{attribute 'linkalways'} 
{attribute 'no_explicit_call' := 'This FB is a CLASS and must be accessed using methods or properties'}
{attribute 'enable_dynamic_creation'}
FUNCTION_BLOCK FINAL NE_DINT EXTENDS Node
VAR
	in1 : _DINT(0);
	in2 : _DINT(0);
	out : _BOOL(FALSE);
END_VAR

METHOD PUBLIC Clone : I_Node
VAR
	pNode : POINTER TO NE_DINT;
END_VAR
pNode := __NEW(NE_DINT);
Clone := pNode^;
END_METHOD

METHOD FB_init : BOOL
VAR_INPUT
	bInitRetains : BOOL; // if TRUE, the retain variables are initialized (warm start / cold start)
	bInCopyCode : BOOL;  // if TRUE, the instance afterwards gets moved into the copy code (online change)
END_VAR
AddInput('in1',THIS^.in1);
AddInput('in2',THIS^.in2);
AddOutput('out', THIS^.out);
END_METHOD

METHOD PROTECTED OnExecute
VAR
END_VAR
out.Value := in1.Value <> in2.Value;
END_METHOD

END_FUNCTION_BLOCK

(* stored: Version 1.1.0.1, ProductVersion 3.1.4024.15
   POU NE_DINT: Id {dc90bf6d-96e3-4071-902f-2370f234dd21}, SpecialFunc None
   Folder Constructor: Id {d7f0702d-e194-47fb-881f-41a2618626ac}
   Method Clone: Id {36dd97a9-336b-4d01-b38c-7519a4627c73}
   Method FB_init: Id {144253cf-c65d-4f4d-85a0-900d1574b2b7}
   Method OnExecute: Id {c01c01c3-e98a-4e89-9984-31ef3f6cbbc0} *)
